(* Logix 5000 project; controller NSH_PLC1 vendor 1 type 14 code 167 rev 32.11; software revision 32.02 *)
// North State Hulling, PLC #1. Performes all System Logic and communicates with MCC#1, All Flex IO & PLC#2 (MCC#2 & #3)

TASK MainTask (continuous, watchdog 500 ms) : MainProgram, BagHouses, PreClean, HullerSheller

MODULES
   Local : vendor 1 type 14 code 167 (ICP 0, Ethernet 192.168.1.250, rev 32.11)
      AOP_BH1A : PowerFlex 755-EENET (Ethernet 192.168.0.41, rev 14.4, Output RPI 250 ms)   // Baghouse #1 Fan
          : vendor 1 type 143 code 32928 (RhinoBP 13, rev 1.1)
          : vendor 1 type 143 code 33184 (RhinoBP 14, rev 2.5)
      AOP_H28_D : PowerFlex 525-EENET (Ethernet 192.168.1.56, rev 6.1, Output RPI 250 ms)   // Nolan Shear Roll
      AOP_Local_Flex_IO : 1794-AENTR (Ethernet 192.168.0.32, rev 1.1, Output RPI 250 ms)   // PLC Panel Flex IO
         Input_L1 : 1794-IA16 (Flex 0, rev 1.1)
         Output_L6 : vendor 1 type 7 code 48 (Flex 5, rev 1.1)
         Input_L4 : 1794-IA16 (Flex 3, rev 1.1)
         Input_L5 : 1794-IA16 (Flex 4, rev 1.1)
         Input_L2 : 1794-IA16 (Flex 1, rev 1.1)
         Input_L3 : 1794-IA16 (Flex 2, rev 1.1)
         Output_L7 : vendor 1 type 7 code 48 (Flex 6, rev 1.1)
         Output_L8 : vendor 1 type 7 code 48 (Flex 7, rev 1.1)
      AOP_Remote_Flex_IO : 1794-AENTR (Ethernet 192.168.0.51, rev 1.1, Output RPI 250 ms)   // Remote Flex IO
         Input_R1 : 1794-IA16 (Flex 0, rev 1.1)
         Input_R2 : 1794-IA16 (Flex 1, rev 1.1)
         Input_R3 : 1794-IA16 (Flex 2, rev 1.1)
         Input_R4 : 1794-IA16 (Flex 3, rev 1.1)
         Input_R5 : 1794-IA16 (Flex 4, rev 1.1)
         Output_R6 : vendor 1 type 7 code 48 (Flex 5, rev 1.1)
         Output_R7 : vendor 1 type 7 code 48 (Flex 6, rev 1.1)
         Output_R8 : vendor 1 type 7 code 48 (Flex 7, rev 1.1)
      AOP_P_9A : 193-ECM-ETR (Ethernet 192.168.1.45, rev 7.1, StandardDataDriven RPI 250 ms)
END_MODULES

TYPE MainBins :   // Main Bins, Gates, Switches and Bindicators
STRUCT
   SW_A_Opened : BOOL;   // Line 1, Bin Gate Opened Switch
   SW_A_Closed : BOOL;   // Line 1, Bin Gate Closed Switch
   SV_Open_A : BOOL;   // Line 1, Open Bin Gate Soleniod
   SW_B_Opened : BOOL;   // Line 2, Bin Gate Opened Switch
   SW_B_Closed : BOOL;   // Line 2, Bin Gate Closed Switch
   SV_Open_B : BOOL;   // Line 2, Open Bin Gate Soleniod
   BN_Full : BOOL;   // Bin Full Bindicator
   TMR_BinFull : TIMER;   // Bin is Full TON Timer
   TMR_BinNotFull : TIMER;   // Bin is Not Full TON Timer
   LT_FullVisible : BOOL;   // HMI Bin Full Light, Visible
   LT_FullFlash : BOOL;   // HMI Bin Full Light, Flash
   MSG_Status_A : DINT;   // 0=Closed (Red) 1=Opened (Green) 2=Inbetween (Flash Yellow)
   MSG_Status_B : DINT;   // 0=Closed (Red) 1=Opened (Green) 2=Inbetween (Flash Yellow)
END_STRUCT
END_TYPE

TYPE Motor :
STRUCT
   StatusBits : DINT;   // Status Bits
   Run : BOOL;   // Run Motor
   Running : BOOL;   // Motor is Running
   NextMotorOK : BOOL;   // Ok, Run Next Motor
   Run_TON : TIMER;   // Running + Time, Run Next Motor
   Amps : REAL;   // Amps
   MSG_GraphicsState : DINT;   // 0=Red 1=Grn 2=FlashYel 3=FlashBlue 4=FlashRed
   HandAuto : BOOL;   // Radio Buttons, On=Hand, Off=Auto
   RunStop : BOOL;   // Pushbuttons, On=Run, Off=Stop
   Fault : BOOL;   // On=Fault
   Fault_TON : TIMER;   // Delay Before Fault
   Warning : BOOL;   // On=Warning
   Warning_TON : TIMER;   // Delay Before Warning
   MSG_FaultWarning : DINT;   // Display of Fault or Warning Number
   Reset_TOF : TIMER;   // Fault Reset Duration to Drive
   HandAuto_OSB : BOOL;   // Radio Buttons HandAuto Transition Relay
   DD_OverloadPercent : DINT;   // Overload 0.0-100.0%, Data Display
   StopTimer : TIMER;   // Shutdown Stop Timer
END_STRUCT
END_TYPE

TYPE VFD_Extra :
STRUCT
   DE_Speed : DINT;   // Speed, 1-100%, Data Entry
   DD_SpeedFactored : DINT;   // Speed, (1-100%, X Factor) Data Display
   DE_OverloadPercent : DINT;   // Overload Warning 1-100%, Data Entry
END_STRUCT
END_TYPE

VAR_GLOBAL   (* controller tags *)
   AFI : BOOL;   // Always False
   BH1 : Motor := (Run_TON.PRE := 1500, StopTimer.PRE := 1500);   // Auger
   BH1A : Motor := (Run_TON.PRE := 1500, StopTimer.PRE := 1500);   // Fan
   BH1A_VFD : VFD_Extra;   // Fan
   BH1B : Motor := (Run_TON.PRE := 1500, StopTimer.PRE := 1500);   // Rev.Fan
   BH1C : Motor := (Run_TON.PRE := 1500, StopTimer.PRE := 1500);   // Rev. Arm
   BH1D : Motor := (Run_TON.PRE := 1500, StopTimer.PRE := 1500);   // Airlock
   BH2 : Motor := (Run_TON.PRE := 1500, StopTimer.PRE := 1500);   // S. Ele
   BH2A : Motor := (Run_TON.PRE := 1500, StopTimer.PRE := 1500);   // Fan
   BH2A_VFD : VFD_Extra;   // Fan
   BH2B : Motor := (Run_TON.PRE := 1500, StopTimer.PRE := 1500);   // Rev.Fan
   BH2C : Motor := (Run_TON.PRE := 1500, StopTimer.PRE := 1500);   // Rev. Arm
   BH2D : Motor := (Run_TON.PRE := 1500);   // Airlock
   BH3 : Motor := (Run_TON.PRE := 1500, StopTimer.PRE := 1500);   // BH Rock
   BH3A : Motor := (Run_TON.PRE := 1500, StopTimer.PRE := 1500);   // Fan
   BH3A_VFD : VFD_Extra;   // Fan
   BH3B : Motor := (Run_TON.PRE := 1500, StopTimer.PRE := 1500);   // Rev.Fan
   BH3C : Motor := (Run_TON.PRE := 1500, StopTimer.PRE := 1500);   // Rev. Arm
   BH3D : Motor := (Run_TON.PRE := 1500, StopTimer.PRE := 1500);   // Airlock
   BH_FansStarting : BOOL;   // Baghouse 1, 2 or 3 Fans Starting
   C10 : Motor := (Run_TON.PRE := 1500, StopTimer.PRE := 1500);   // Auger
   C1A : Motor := (Run_TON.PRE := 1500, StopTimer.PRE := 1500);   // Auger
   C1B : Motor := (Run_TON.PRE := 1500, StopTimer.PRE := 1500);   // Auger
   C2 : Motor := (Run_TON.PRE := 1500, StopTimer.PRE := 1500);   // Auger
   C3A : Motor := (Run_TON.PRE := 1500, StopTimer.PRE := 1500);   // Auger
   C3B : Motor := (Run_TON.PRE := 1500, StopTimer.PRE := 1500);   // Auger
   C4 : Motor := (Run_TON.PRE := 1500, StopTimer.PRE := 1500);   // Ele.
   C5 : Motor := (Run_TON.PRE := 1500);   // Aspirator
   C7 : Motor := (Run_TON.PRE := 1500, StopTimer.PRE := 1500);   // Ele
   C8 : Motor := (Run_TON.PRE := 1500, StopTimer.PRE := 1500);   // Auger
   C9 : Motor := (Run_TON.PRE := 1500, StopTimer.PRE := 1500);   // Auger
   CL1 : Motor := (Run_TON.PRE := 1500, StopTimer.PRE := 1500);   // Auger
   CL2 : Motor := (Run_TON.PRE := 1500, StopTimer.PRE := 1500);   // Auger
   CL3 : Motor := (Run_TON.PRE := 1500, StopTimer.PRE := 1500);   // Auger
   CL4 : Motor := (Run_TON.PRE := 1500, StopTimer.PRE := 1500);   // Auger
   CL5 : Motor := (Run_TON.PRE := 1500, StopTimer.PRE := 1500);   // Auger
   CL6 : Motor := (Run_TON.PRE := 1500, StopTimer.PRE := 1500);   // Auger
   CR_LastBH1Fan : BOOL;   // Last Motor in Baghouse 1 Fans Running
   CR_LastBH2Fan : BOOL;   // Last Motor in Baghouse 2 Fans Running
   CR_LastBH3Fan : BOOL;   // Last Motor in Baghouse 3 Fans Running
   CR_LastLine1 : BOOL;   // Last Motor in line 1 Running
   CR_LastLine2 : BOOL;   // Last Motor in line 2 Running
   CR_LastPC1Fan : BOOL;   // Last Motor in Line 1 Fans Running
   CR_LastPC2Fan : BOOL;   // Last Motor in Line 2 Fans Running
   CR_RunBH2_Fans : BOOL;   // Run Baghouse 2 Fans Relay
   CR_RunBH2_FansCO : BOOL;   // Run Baghouse 2 Fans Cleanout Relay
   CR_RunBH3_Fans : BOOL;   // Run Baghouse 3 Fans Relay
   CR_RunBH3_FansCO : BOOL;   // Run Baghouse 3 Fans Cleanout Relay
   CR_RunBH_Fans : BOOL;   // Run Baghouse's Fans Relay
   CR_RunBH_FansCO : BOOL;   // Run Baghouse's Cleanout Relay
   CR_RunCommon : BOOL;   // PreClean, Run Common Units
   CR_RunHS : BOOL;   // Run Hullers & Shellers Relay
   CR_RunHullerShellers : BOOL;   // Run Hullers & Shellers
   CR_RunLine1 : BOOL;   // Pre Clean Run Line 1 Relay
   CR_RunLine2 : BOOL;   // Pre Clean Run Line 2 Relay
   CR_RunPC1_Fans : BOOL;   // Pre Clean Run Line 1 Fans Relay
   CR_RunPC1_FansCO : BOOL;   // Pre Clean Run Line 1 Fans Cleanout Relay
   CR_RunPC2_Fans : BOOL;   // Pre Clean Run Line 2 Fans Relay
   CR_RunPC2_FansCO : BOOL;   // Pre Clean Run Line 2 Fans Cleanout Relay
   CR_StopBH_Fans : BOOL;   // Stop Baghouse's Fans Relay
   CR_StopBH_FansCO : BOOL;   // Stop Baghouse's Fans Cleanout Relay
   CR_StopCommon : BOOL;   // PreClean, Stop Common Units
   CR_StopHS : BOOL;   // Stop Hullers & Shellers Relay
   CR_StopLine1 : BOOL;   // Pre Clean Stop Line 1 Relay
   CR_StopLine2 : BOOL;   // Pre Clean Stop Line 2 Relay
   CR_StopPC1_Fans : BOOL;   // Pre Clean Stop Line 1 Fans Relay
   CR_StopPC1_FansCO : BOOL;   // Pre Clean Stop Line 1 Fans Cleanout Relay
   CR_StopPC2_Fans : BOOL;   // Pre Clean Stop Line 2 Fans Relay
   CR_StopPC2_FansCO : BOOL;   // Pre Clean Stop Line 2 Fans Cleanout Relay
   D10 : Motor := (Run_TON.PRE := 1500, StopTimer.PRE := 1500);   // Ele
   D11 : Motor := (Run_TON.PRE := 1500, StopTimer.PRE := 1500);   // Auger
   D12 : Motor := (Run_TON.PRE := 1500, StopTimer.PRE := 1500);   // Auger
   D13 : Motor := (Run_TON.PRE := 1500, StopTimer.PRE := 1500);   // Auger
   D14 : Motor := (Run_TON.PRE := 1500, StopTimer.PRE := 1500);   // Auger
   D1A : Motor := (Run_TON.PRE := 1500, StopTimer.PRE := 1500);   // Auger
   D1B : Motor := (Run_TON.PRE := 1500, StopTimer.PRE := 1500);   // Auger
   D2 : Motor := (Run_TON.PRE := 1500, StopTimer.PRE := 1500);   // Auger
   D3 : Motor := (Run_TON.PRE := 1500);   // Aspirator
   D4 : Motor := (Run_TON.PRE := 1500, StopTimer.PRE := 1500);   // Auger
   D5 : Motor := (Run_TON.PRE := 1500, StopTimer.PRE := 1500);   // Auger
   D6 : Motor := (Run_TON.PRE := 1500, StopTimer.PRE := 1500);   // Auger
   D7 : Motor := (Run_TON.PRE := 1500);   // Aspirator
   DE_PC_MasterSpeedFactor : DINT;   // PreClean Master Speed Factor 75%->125%
   DL1 : Motor := (Run_TON.PRE := 1500, StopTimer.PRE := 1500);   // Auger
   DummyLastMotor : BOOL;   // Last Motor in Start Sequence
   DummyOutput : BOOL;
   DummyVFD : VFD_Extra;   // Dummy
   H1 : Motor := (Run_TON.PRE := 1500, StopTimer.PRE := 1500);   // Conv.
   H10 : Motor := (Run_TON.PRE := 1500, StopTimer.PRE := 1500);   // Auger
   H11 : Motor := (Run_TON.PRE := 1500, StopTimer.PRE := 1500);   // Ele.
   H12 : Motor := (Run_TON.PRE := 1500, StopTimer.PRE := 1500);   // Auger
   H13 : Motor := (Run_TON.PRE := 1500, StopTimer.PRE := 1500);   // Auger
   H14A : Motor := (Run_TON.PRE := 1500, StopTimer.PRE := 1500);   // Shr. Roll
   H14B : Motor := (Run_TON.PRE := 1500, StopTimer.PRE := 1500);   // Shr. Roll
   H14C : Motor := (Run_TON.PRE := 1500, StopTimer.PRE := 1500);   // Vib.
   H15A : Motor := (Run_TON.PRE := 1500, StopTimer.PRE := 1500);   // Aspirator
   H15B : Motor := (Run_TON.PRE := 1500, StopTimer.PRE := 1500);   // Aspirator
   H16 : Motor := (Run_TON.PRE := 1500, StopTimer.PRE := 1500);   // Auger
   H17 : Motor := (Run_TON.PRE := 1500, StopTimer.PRE := 1500);   // Roll Fd.
   H18A : Motor := (Run_TON.PRE := 1500, StopTimer.PRE := 1500);   // Shr. Roll
   H18B : Motor := (Run_TON.PRE := 1500, StopTimer.PRE := 1500);   // Shr. Roll
   H18C : Motor := (Run_TON.PRE := 1500, StopTimer.PRE := 1500);   // Vib.
   H19A : Motor := (Run_TON.PRE := 1500, StopTimer.PRE := 1500);   // Aspirator
   H19B : Motor := (Run_TON.PRE := 1500, StopTimer.PRE := 1500);   // Aspirator
   H20A : Motor := (Run_TON.PRE := 1500, StopTimer.PRE := 1500);   // Shr. Roll
   H20B : Motor := (Run_TON.PRE := 1500, StopTimer.PRE := 1500);   // Shr. Roll
   H20C : Motor := (Run_TON.PRE := 1500, StopTimer.PRE := 1500);   // Vib.
   H21A : Motor := (Run_TON.PRE := 1500, StopTimer.PRE := 1500);   // Aspirator
   H21B : Motor := (Run_TON.PRE := 1500, StopTimer.PRE := 1500);   // Aspirator
   H22 : Motor := (Run_TON.PRE := 1500, StopTimer.PRE := 1500);   // BMM
   H22B : Motor := (Run_TON.PRE := 1500);   // Hard Crkr.
   H23A : Motor := (Run_TON.PRE := 1500, StopTimer.PRE := 1500);   // Aspirator
   H23B : Motor := (Run_TON.PRE := 1500, StopTimer.PRE := 1500);   // Aspirator
   H24A : Motor := (Run_TON.PRE := 1500, StopTimer.PRE := 1500);   // Aspirator
   H24B : Motor := (Run_TON.PRE := 1500, StopTimer.PRE := 1500);   // Aspirator
   H25 : Motor := (Run_TON.PRE := 1500, StopTimer.PRE := 1500);   // Ele.
   H26 : Motor := (Run_TON.PRE := 1500, StopTimer.PRE := 1500);   // Auger
   H27 : Motor := (Run_TON.PRE := 1500, StopTimer.PRE := 1500);   // Auger
   H28A : Motor := (Run_TON.PRE := 1500, StopTimer.PRE := 1500);   // HC Vib.
   H28B : Motor := (Run_TON.PRE := 1500, StopTimer.PRE := 1500);   // Hard Crkr.
   H28C : Motor := (Run_TON.PRE := 1500, StopTimer.PRE := 1500);   // S.Roll
   H28D : Motor := (Run_TON.PRE := 1500, StopTimer.PRE := 1500);   // Shr.Roll.
   H29A : Motor := (Run_TON.PRE := 1500, StopTimer.PRE := 1500);   // Aspirator
   H29B : Motor := (Run_TON.PRE := 1500, StopTimer.PRE := 1500);   // Aspirator
   H30 : Motor := (Run_TON.PRE := 1500, StopTimer.PRE := 1500);   // Auger
   H31 : Motor := (Run_TON.PRE := 1500, StopTimer.PRE := 1500);   // Roll Fdr.
   H32A : Motor := (Run_TON.PRE := 1500, StopTimer.PRE := 1500);   // HS Cracker
   H32B : Motor := (Run_TON.PRE := 1500, StopTimer.PRE := 1500);   // Hard Crkr.
   H32C : Motor := (Run_TON.PRE := 1500, StopTimer.PRE := 1500);   // Shr.Roll.
   H32D : Motor := (Run_TON.PRE := 1500, StopTimer.PRE := 1500);   // Shr.Roll.
   H33A : Motor := (Run_TON.PRE := 1500, StopTimer.PRE := 1500);   // Aspirator
   H33B : Motor := (Run_TON.PRE := 1500, StopTimer.PRE := 1500);   // Aspirator
   H34A : Motor := (Run_TON.PRE := 1500, StopTimer.PRE := 1500);   // HC Vib.
   H34B : Motor := (Run_TON.PRE := 1500, StopTimer.PRE := 1500);   // Hard Crkr.
   H34C : Motor := (Run_TON.PRE := 1500, StopTimer.PRE := 1500);   // S.Roll
   H34D : Motor := (Run_TON.PRE := 1500, StopTimer.PRE := 1500);   // Shr.Roll.
   H35A : Motor := (Run_TON.PRE := 1500, StopTimer.PRE := 1500);   // Aspirator
   H35B : Motor := (Run_TON.PRE := 1500, StopTimer.PRE := 1500);   // Aspirator
   H36 : Motor := (Run_TON.PRE := 1500, StopTimer.PRE := 1500);   // BMM
   H37A : Motor := (Run_TON.PRE := 1500, StopTimer.PRE := 1500);   // Aspirator
   H37B : Motor := (Run_TON.PRE := 1500, StopTimer.PRE := 1500);   // Aspirator
   H38A : Motor := (Run_TON.PRE := 1500, StopTimer.PRE := 1500);   // Aspirator
   H38B : Motor := (Run_TON.PRE := 1500, StopTimer.PRE := 1500);   // Aspirator
   H39 : Motor := (Run_TON.PRE := 1500, StopTimer.PRE := 1500);   // Ele.
   H3A : Motor := (Run_TON.PRE := 1500, StopTimer.PRE := 1500);   // Incline
   H3B : Motor := (Run_TON.PRE := 1500, StopTimer.PRE := 1500);   // Ele.
   H4 : Motor := (Run_TON.PRE := 1500, StopTimer.PRE := 1500);   // Auger
   H40 : Motor := (Run_TON.PRE := 1500, StopTimer.PRE := 1500);   // Auger
   H41 : Motor := (Run_TON.PRE := 1500, StopTimer.PRE := 1500);   // Auger
   H42A : Motor := (Run_TON.PRE := 1500, StopTimer.PRE := 1500);   // HC Vib.
   H42B : Motor := (Run_TON.PRE := 1500, StopTimer.PRE := 1500);   // Hard Crkr.
   H42C : Motor := (Run_TON.PRE := 1500, StopTimer.PRE := 1500);   // S.Roll
   H42D : Motor := (Run_TON.PRE := 1500, StopTimer.PRE := 1500);   // Shr.Roll.
   H42H : Motor := (Run_TON.PRE := 1500);   // Auger
   H43A : Motor := (Run_TON.PRE := 1500, StopTimer.PRE := 1500);   // Aspirator
   H43B : Motor := (Run_TON.PRE := 1500, StopTimer.PRE := 1500);   // Aspirator
   H44A : Motor := (Run_TON.PRE := 1500, StopTimer.PRE := 1500);   // HC Vib.
   H44B : Motor := (Run_TON.PRE := 1500, StopTimer.PRE := 1500);   // Hard Crkr.
   H44C : Motor := (Run_TON.PRE := 1500, StopTimer.PRE := 1500);   // S.Roll
   H44D : Motor := (Run_TON.PRE := 1500, StopTimer.PRE := 1500);   // Shr.Roll.
   H45A : Motor := (Run_TON.PRE := 1500, StopTimer.PRE := 1500);   // Aspirator
   H45B : Motor := (Run_TON.PRE := 1500, StopTimer.PRE := 1500);   // Aspirator
   H46 : Motor := (Run_TON.PRE := 1500, StopTimer.PRE := 1500);   // BMM
   H47A : Motor := (Run_TON.PRE := 1500, StopTimer.PRE := 1500);   // Aspirator
   H47B : Motor := (Run_TON.PRE := 1500, StopTimer.PRE := 1500);   // Aspirator
   H48A : Motor := (Run_TON.PRE := 1500, StopTimer.PRE := 1500);   // Aspirator
   H48B : Motor := (Run_TON.PRE := 1500, StopTimer.PRE := 1500);   // Aspirator
   H49 : Motor := (Run_TON.PRE := 1500, StopTimer.PRE := 1500);   // Ele.
   H5 : Motor := (Run_TON.PRE := 1500, StopTimer.PRE := 1500);   // Auger
   H50A : Motor := (Run_TON.PRE := 1500, StopTimer.PRE := 1500);   // Auger
   H50B : Motor := (Run_TON.PRE := 1500, StopTimer.PRE := 1500);   // Auger
   H6 : Motor := (Run_TON.PRE := 1500, StopTimer.PRE := 1500);   // Roll Fd.
   H7 : Motor := (Run_TON.PRE := 1500, StopTimer.PRE := 1500);   // BMM
   H8A : Motor := (Run_TON.PRE := 1500, StopTimer.PRE := 1500);   // Aspirator
   H8B : Motor := (Run_TON.PRE := 1500, StopTimer.PRE := 1500);   // Aspirator
   H9A : Motor := (Run_TON.PRE := 1500, StopTimer.PRE := 1500);   // Aspirator
   H9B : Motor := (Run_TON.PRE := 1500, StopTimer.PRE := 1500);   // Aspirator
   HS_Horn : BOOL;   // Huller Sheller, Horn Output
   HS_LastMotor : BOOL;   // Last Motor in Huller Sheller Sequence is Running
   HS_NoEstops : BOOL;   // Huller Sheller, No Estops
   HS_Starting : BOOL;   // Sheller Sequence is Starting, Prevent Preclean from Starting
   LS101 : BOOL;   // Dummy Limit Switch
   M10 : Motor := (Run_TON.PRE := 1500, StopTimer.PRE := 1500);   // Vib.
   M10A : Motor := (Run_TON.PRE := 1500, StopTimer.PRE := 1500);   // Asp.
   M10B : Motor := (Run_TON.PRE := 1500, StopTimer.PRE := 1500);   // Asp.
   M11 : Motor := (Run_TON.PRE := 1500, StopTimer.PRE := 1500);   // Ele.
   M12aA : Motor := (Run_TON.PRE := 1500, StopTimer.PRE := 1500);   // Grav.Sep
   M12aB : Motor := (Run_TON.PRE := 1500, StopTimer.PRE := 1500);   // Syntron
   M13aA : Motor := (Run_TON.PRE := 1500, StopTimer.PRE := 1500);   // Grav.Sep
   M13aB : Motor := (Run_TON.PRE := 1500, StopTimer.PRE := 1500);   // Syntron
   M14 : Motor := (Run_TON.PRE := 1500, StopTimer.PRE := 1500);   // Vib.
   M15 : Motor := (Run_TON.PRE := 1500, StopTimer.PRE := 1500);   // Ele.
   M16 : Motor := (Run_TON.PRE := 1500, StopTimer.PRE := 1500);   // Evo.
   M16R : Motor;   // Conveyor
   M17 : Motor := (Run_TON.PRE := 1500, StopTimer.PRE := 1500);   // Evo.
   M18 : Motor := (Run_TON.PRE := 1500, StopTimer.PRE := 1500);   // Vib.
   M19 : Motor := (Run_TON.PRE := 1500, StopTimer.PRE := 1500);   // Ele.
   M1A : Motor := (Run_TON.PRE := 1500, StopTimer.PRE := 1500);   // Vib.
   M2 : Motor := (Run_TON.PRE := 1500, StopTimer.PRE := 1500);   // Vib.
   M20 : Motor := (Run_TON.PRE := 1500, StopTimer.PRE := 1500);   // Ele.
   M21 : Motor := (Run_TON.PRE := 1500, StopTimer.PRE := 1500);   // Nolin
   M25 : Motor := (Run_TON.PRE := 1500, StopTimer.PRE := 1500);   // Accept Vib.
   M27 : Motor := (Run_TON.PRE := 1500, StopTimer.PRE := 1500);   // Belt
   M28 : Motor := (Run_TON.PRE := 1500, StopTimer.PRE := 1500);   // Belt
   M29 : Motor := (Run_TON.PRE := 1500, StopTimer.PRE := 1500);   // Ele.
   M3 : Motor := (Run_TON.PRE := 1500, StopTimer.PRE := 1500);   // Belt
   M30A : Motor := (Run_TON.PRE := 1500, StopTimer.PRE := 1500);   // HC Vib.
   M30B : Motor := (Run_TON.PRE := 1500, StopTimer.PRE := 1500);   // Hard Crkr.
   M30C : Motor := (Run_TON.PRE := 1500, StopTimer.PRE := 1500);   // Shr.Roll.
   M30D : Motor := (Run_TON.PRE := 1500, StopTimer.PRE := 1500);   // Shr.Roll.
   M31A : Motor := (Run_TON.PRE := 1500, StopTimer.PRE := 1500);   // Asp.
   M31B : Motor := (Run_TON.PRE := 1500, StopTimer.PRE := 1500);   // Asp.
   M32A : Motor := (Run_TON.PRE := 1500, StopTimer.PRE := 1500);   // Vib.Scrn.
   M32B : Motor := (Run_TON.PRE := 1500, StopTimer.PRE := 1500);   // Ele.
   M33 : Motor := (Run_TON.PRE := 1500, StopTimer.PRE := 1500);   // Belt
   M34 : Motor := (Run_TON.PRE := 1500, StopTimer.PRE := 1500);   // Destoner
   M35 : Motor := (Run_TON.PRE := 1500, StopTimer.PRE := 1500);   // Ele.
   M36A : Motor := (Run_TON.PRE := 1500, StopTimer.PRE := 1500);   // G. Sep.
   M36B : Motor := (Run_TON.PRE := 1500, StopTimer.PRE := 1500);   // R. Feeder.
   M37 : Motor := (Run_TON.PRE := 1500, StopTimer.PRE := 1500);   // 5x12
   M38A : Motor := (Run_TON.PRE := 1500, StopTimer.PRE := 1500);   // Asp.
   M38B : Motor := (Run_TON.PRE := 1500, StopTimer.PRE := 1500);   // Asp.
   M39 : Motor := (Run_TON.PRE := 1500, StopTimer.PRE := 1500);   // Ele.
   M391 : Motor := (Run_TON.PRE := 1500);   // Ele.
   M4 : Motor := (Run_TON.PRE := 1500, StopTimer.PRE := 1500);   // Vib.
   M40A : Motor := (Run_TON.PRE := 1500, StopTimer.PRE := 1500);   // Sep.
   M40B : Motor := (Run_TON.PRE := 1500, StopTimer.PRE := 1500);   // Syn.Fer.
   M41 : Motor := (Run_TON.PRE := 1500, StopTimer.PRE := 1500);   // Ele.
   M42C : Motor := (Run_TON.PRE := 1500, StopTimer.PRE := 1500);   // 3C Deck
   M42D : Motor := (Run_TON.PRE := 1500, StopTimer.PRE := 1500);   // 3C Deck
   M43CA : Motor := (Run_TON.PRE := 1500, StopTimer.PRE := 1500);   // Asp.
   M43CB : Motor := (Run_TON.PRE := 1500, StopTimer.PRE := 1500);   // Asp.
   M43DA : Motor := (Run_TON.PRE := 1500, StopTimer.PRE := 1500);   // Asp.
   M43DB : Motor := (Run_TON.PRE := 1500, StopTimer.PRE := 1500);   // Asp.
   M44A : Motor := (Run_TON.PRE := 1500, StopTimer.PRE := 1500);   // Belt
   M44B : Motor := (Run_TON.PRE := 1500, StopTimer.PRE := 1500);   // Belt
   M5 : Motor := (Run_TON.PRE := 1500, StopTimer.PRE := 1500);   // Vib.
   M6 : Motor := (Run_TON.PRE := 1500, StopTimer.PRE := 1500);   // Belt
   M7 : Motor := (Run_TON.PRE := 1500, StopTimer.PRE := 1500);   // Ele.
   M8 : Motor := (Run_TON.PRE := 1500, StopTimer.PRE := 1500);   // Shkr.
   M9A : Motor := (Run_TON.PRE := 1500, StopTimer.PRE := 1500);   // Asp.
   M9B : Motor := (Run_TON.PRE := 1500, StopTimer.PRE := 1500);   // Asp.
   MainBin1 : MainBins;   // PreClean to Huller, Main Bin #1
   MainBin2 : MainBins;   // PreClean to Huller, Main Bin #1
   MainBin3 : MainBins;   // PreClean to Huller, Main Bin #1
   MainBin4 : MainBins;   // PreClean to Huller, Main Bin #1
   MainBin5 : MainBins;   // PreClean to Huller, Main Bin #1
   MainBin6 : MainBins;   // PreClean to Huller, Main Bin #1
   MainBin7 : MainBins;   // PreClean to Huller, Main Bin #1
   MainBin8 : MainBins;   // PreClean to Huller, Main Bin #1
   NewWarning : BOOL;   // New Huller-Sheller Warning has just occured
   Num_Warning_LS : DINT;   // Number of Warnings Last Scan, Detect New
   P10_5A : Motor := (Run_TON.PRE := 1500, StopTimer.PRE := 1500);   // Cross Auger
   P10_5B : Motor := (Run_TON.PRE := 1500, StopTimer.PRE := 1500);   // Cross Auger
   P10A : Motor := (Run_TON.PRE := 1500, StopTimer.PRE := 1500);   // Elev to Bins
   P10B : Motor := (Run_TON.PRE := 1500, StopTimer.PRE := 1500);   // Elev to Bins
   P11A : Motor := (Run_TON.PRE := 1500, StopTimer.PRE := 1500);   // Line1 Auger
   P11B : Motor := (Run_TON.PRE := 1500, StopTimer.PRE := 1500);   // Line2 Auger
   P1A : Motor := (Run_TON.PRE := 1500, StopTimer.PRE := 1500);   // DO Conv.
   P1B : Motor := (Run_TON.PRE := 1500, StopTimer.PRE := 1500);   // Auger
   P2A : Motor := (Run_TON.PRE := 1500, StopTimer.PRE := 1500);   // Cross Conv.
   P2B : Motor := (Run_TON.PRE := 1500, StopTimer.PRE := 1500);   // Stick Reel
   P3A : Motor := (Run_TON.PRE := 1500, StopTimer.PRE := 1500);   // Stick Reel
   P3B : Motor := (Run_TON.PRE := 1500, StopTimer.PRE := 1500);   // Stick Reel
   P4A : Motor := (Run_TON.PRE := 1500, StopTimer.PRE := 1500);   // C. Belt
   P4B : Motor := (Run_TON.PRE := 1500, StopTimer.PRE := 1500);   // C. Belt
   P5A : Motor := (Run_TON.PRE := 1500, StopTimer.PRE := 1500);   // Ele. to Vib
   P5B : Motor := (Run_TON.PRE := 1500, StopTimer.PRE := 1500);   // Ele. to Vib
   P6A : Motor := (Run_TON.PRE := 1500, StopTimer.PRE := 1500);   // Vib Splitter
   P6B : Motor := (Run_TON.PRE := 1500, StopTimer.PRE := 1500);   // Vib.Spltr.
   P7A : Motor := (Run_TON.PRE := 1500, StopTimer.PRE := 1500);   // Screener
   P7A1 : Motor := (Run_TON.PRE := 1500);   // Screener
   P7A2 : Motor := (Run_TON.PRE := 1500, StopTimer.PRE := 1500);   // Screener
   P7B : Motor := (Run_TON.PRE := 1500, StopTimer.PRE := 1500);   // Screener
   P7B2_A : Motor := (Run_TON.PRE := 1500, StopTimer.PRE := 1500);   // Screener
   P7B2_B : Motor := (Run_TON.PRE := 1500, StopTimer.PRE := 1500);   // Rot.Fdr.
   P8A2_A : Motor := (Run_TON.PRE := 1500, StopTimer.PRE := 1500);   // Destoner
   P8A2_B : Motor := (Run_TON.PRE := 1500, StopTimer.PRE := 1500);   // AirLock
   P8A_A : Motor := (Run_TON.PRE := 1500, StopTimer.PRE := 1500);   // Destoner
   P8A_B : Motor := (Run_TON.PRE := 1500, StopTimer.PRE := 1500);   // Airlock
   P8B : Motor := (Run_TON.PRE := 1500, StopTimer.PRE := 1500);   // Destoner
   P8B2_A : Motor := (Run_TON.PRE := 1500, StopTimer.PRE := 1500);   // Destoner
   P8B2_B : Motor := (Run_TON.PRE := 1500, StopTimer.PRE := 1500);   // Rot.Fdr.
   P9A : Motor := (Run_TON.PRE := 1500, StopTimer.PRE := 1500);   // Auger
   P9B : Motor := (Run_TON.PRE := 1500, StopTimer.PRE := 1500);   // Auger
   PB_HS_Inshell : BOOL;   // Hullers & Shellers Run Inshell Button
   PB_HS_Meats : BOOL;   // Hullers & Shellers Run Meats Button
   PB_HSFaultReset : BOOL;   // Huller Sheller, Fault Reset Button
   PB_PCFaultReset : BOOL;   // PreClean Fault Reset Button
   PB_StartBH_Fans : BOOL;   // Start Baghouse's Fans Button
   PB_StartBH_FansCO : BOOL;   // Start Baghouse's Cleanout Button
   PB_StartHS : BOOL;   // Start Hullers & Shellers Button
   PB_StartLine1 : BOOL;   // Pre Clean Start Line 1 Button
   PB_StartLine2 : BOOL;   // Pre Clean Start Line 2 Button
   PB_StartPC1_Fans : BOOL;   // Pre Clean Start Line 1 Fans Button
   PB_StartPC1_FansCO : BOOL;   // Pre Clean Start Line 1 Fans Cleanout Button
   PB_StartPC2_Fans : BOOL;   // Pre Clean Start Line 2 Fans Button
   PB_StartPC2_FansCO : BOOL;   // Pre Clean Start Line 2 Fans Cleanout Button
   PB_StopBH_Fans : BOOL;   // Stop Baghouse's Fans Button
   PB_StopBH_FansCO : BOOL;   // Stop Baghouse's Fans Cleanout Button
   PB_StopHS : BOOL;   // Stop Hullers & Shellers Button
   PB_StopLine1 : BOOL;   // Pre Clean Stop Line 1 Button
   PB_StopLine2 : BOOL;   // Pre Clean Stop Line 2 Button
   PB_StopPC1_Fans : BOOL;   // Pre Clean Stop Line 1 Fans Button
   PB_StopPC1_FansCO : BOOL;   // Pre Clean Stop Line 1 Fans Cleanout Button
   PB_StopPC2_Fans : BOOL;   // Pre Clean Stop Line 2 Fans Button
   PB_StopPC2_FansCO : BOOL;   // Pre Clean Stop Line 2 Fans Cleanout Button
   PBB1A : Motor := (Run_TON.PRE := 1500, StopTimer.PRE := 1500);   // AirLock
   PBB1B : Motor := (Run_TON.PRE := 1500, StopTimer.PRE := 1500);   // Arm
   PBB1C : Motor := (Run_TON.PRE := 1500, StopTimer.PRE := 1500);   // Cleaning Fan,
   PBB1D : Motor := (Run_TON.PRE := 1500, StopTimer.PRE := 1500);   // Fan,
   PBB1D_VFD : VFD_Extra;   // Fan
   PBB2A : Motor := (Run_TON.PRE := 1500, StopTimer.PRE := 1500);   // AirLock
   PBB2B : Motor := (Run_TON.PRE := 1500, StopTimer.PRE := 1500);   // Arm
   PBB2C : Motor := (Run_TON.PRE := 1500, StopTimer.PRE := 1500);   // Cleaning Fan,
   PBB2D : Motor := (Run_TON.PRE := 1500, StopTimer.PRE := 1500);   // Fan,
   PBL_HS_Inshell : BOOL;   // Hullers & Shellers Run Inshell Button Light
   PBL_HS_Meats : BOOL;   // Hullers & Shellers Run Meats Button Light
   PBL_PCFaultReset : BOOL;   // PreClean Fault Reset Button Light
   PBL_StartBH_Fans : BOOL;   // Start Baghouse's Fans Button Light
   PBL_StartBH_FansCO : BOOL;   // Start Baghouse's Cleanout Button Light
   PBL_StartHS : BOOL;   // Start Hullers & Shellers Button Light
   PBL_StartLine1 : BOOL;   // Pre Clean Start Line 1 Button Light
   PBL_StartLine2 : BOOL;   // Pre Clean Start Line 2 Button Light
   PBL_StartPC1_Fans : BOOL;   // Pre Clean Start Line 1 Fans Button Light
   PBL_StartPC1_FansCO : BOOL;   // Pre Clean Start Line 1 Fans Cleanout Button Light
   PBL_StartPC2_Fans : BOOL;   // Pre Clean Start Line 2 Fans Button Light
   PBL_StartPC2_FansCO : BOOL;   // Pre Clean Start Line 2 Fans Cleanout Button Light
   PBL_StopBH_Fans : BOOL;   // Stop Baghouse's Fans Button Light
   PBL_StopBH_FansCO : BOOL;   // Stop Baghouse's Fans Cleanout Button Light
   PBL_StopHS : BOOL;   // Stop Hullers & Shellers Button Light
   PBL_StopLine1 : BOOL;   // Pre Clean Stop Line 1 Button Light
   PBL_StopLine2 : BOOL;   // Pre Clean Stop Line 2 Button Light
   PBL_StopPC1_Fans : BOOL;   // Pre Clean Stop Line 1 Fans Button Light
   PBL_StopPC1_FansCO : BOOL;   // Pre Clean Stop Line 1 Fans Cleanout Button Light
   PBL_StopPC2_Fans : BOOL;   // Pre Clean Stop Line 2 Fans Button Light
   PBL_StopPC2_FansCO : BOOL;   // Pre Clean Stop Line 2 Fans Cleanout Button Light
   PC_AlarmPulseHorn : BOOL;   // PreClean, New Alarm, Pulse Horn
   PC_FansStarting : BOOL;   // Pre Clean Fans Starting
   PC_FaultResetHorn : BOOL;   // PreClean, Fault Reset, sound Horn
   PC_Horn : BOOL;   // PreClean, Horn Output
   PC_LinesStarting : BOOL;   // Pre Clean Line 1 or 2 Starting
   PC_NoEstops : BOOL;   // PreClean, No Estops
   PD1 : Motor := (Run_TON.PRE := 1500, StopTimer.PRE := 1500);   // Dirt Conv.
   PD2 : Motor := (Run_TON.PRE := 1500, StopTimer.PRE := 1500);   // Incline
   PR1 : Motor := (Run_TON.PRE := 1500, StopTimer.PRE := 1500);   // Rock Conv.
   PR2 : Motor := (Run_TON.PRE := 1500, StopTimer.PRE := 1500);   // Inc. Rock
   PR3 : Motor := (Run_TON.PRE := 1500, StopTimer.PRE := 1500);   // Belt
   PS1 : Motor := (Run_TON.PRE := 1500, StopTimer.PRE := 1500);   // Stick Conv.
   PS2 : Motor := (Run_TON.PRE := 1500, StopTimer.PRE := 1500);   // Inc. Stick Conv.
   PS3 : Motor := (Run_TON.PRE := 1500, StopTimer.PRE := 1500);   // Twig Conv.
   PS4 : Motor := (Run_TON.PRE := 1500, StopTimer.PRE := 1500);   // Twig Conv.
   S1 : Motor := (Run_TON.PRE := 1500, StopTimer.PRE := 1500);   // Vib.
   S10 : Motor := (Run_TON.PRE := 1500, StopTimer.PRE := 1500);   // Auger
   S11 : Motor := (Run_TON.PRE := 1500, StopTimer.PRE := 1500);   // Ele.
   S12 : Motor := (Run_TON.PRE := 1500, StopTimer.PRE := 1500);   // Auger
   S13 : Motor := (Run_TON.PRE := 1500, StopTimer.PRE := 1500);   // Ele.
   S14 : Motor := (Run_TON.PRE := 1500, StopTimer.PRE := 1500);   // Auger
   S15 : Motor := (Run_TON.PRE := 1500, StopTimer.PRE := 1500);   // Auger
   S16A : Motor := (Run_TON.PRE := 1500, StopTimer.PRE := 1500);   // Auger
   S16B : Motor := (Run_TON.PRE := 1500, StopTimer.PRE := 1500);   // Auger
   S17A : Motor := (Run_TON.PRE := 1500, StopTimer.PRE := 1500);   // HS Cracker
   S17B : Motor := (Run_TON.PRE := 1500, StopTimer.PRE := 1500);   // Hard Crkr.
   S17C : Motor := (Run_TON.PRE := 1500, StopTimer.PRE := 1500);   // Shr.Roll.
   S17D : Motor := (Run_TON.PRE := 1500, StopTimer.PRE := 1500);   // S.Roll
   S18A : Motor := (Run_TON.PRE := 1500, StopTimer.PRE := 1500);   // HC Vib.
   S18B : Motor := (Run_TON.PRE := 1500, StopTimer.PRE := 1500);   // Hard Crkr.
   S18C : Motor := (Run_TON.PRE := 1500, StopTimer.PRE := 1500);   // Shr.Roll.
   S18D : Motor := (Run_TON.PRE := 1500, StopTimer.PRE := 1500);   // S.Roll
   S19 : Motor := (Run_TON.PRE := 1500, StopTimer.PRE := 1500);   // Gry.
   S2 : Motor := (Run_TON.PRE := 1500, StopTimer.PRE := 1500);   // Ele.
   S20 : Motor := (Run_TON.PRE := 1500, StopTimer.PRE := 1500);   // Ele.
   S21 : Motor := (Run_TON.PRE := 1500, StopTimer.PRE := 1500);   // Roll Fdr.
   S22A : Motor := (Run_TON.PRE := 1500, StopTimer.PRE := 1500);   // HC Vib.
   S22B : Motor := (Run_TON.PRE := 1500, StopTimer.PRE := 1500);   // Hard Crkr.
   S22C : Motor := (Run_TON.PRE := 1500, StopTimer.PRE := 1500);   // Shr.Roll.
   S22D : Motor := (Run_TON.PRE := 1500, StopTimer.PRE := 1500);   // S.Roll
   S23A : Motor := (Run_TON.PRE := 1500, StopTimer.PRE := 1500);   // HC Vib.
   S23B : Motor := (Run_TON.PRE := 1500, StopTimer.PRE := 1500);   // Hard Crkr.
   S23C : Motor := (Run_TON.PRE := 1500, StopTimer.PRE := 1500);   // Shr.Roll.
   S23D : Motor := (Run_TON.PRE := 1500, StopTimer.PRE := 1500);   // S.Roll
   S24 : Motor := (Run_TON.PRE := 1500, StopTimer.PRE := 1500);   // Deck
   S25 : Motor := (Run_TON.PRE := 1500, StopTimer.PRE := 1500);   // Ele.
   S26 : Motor := (Run_TON.PRE := 1500, StopTimer.PRE := 1500);   // Auger
   S27 : Motor := (Run_TON.PRE := 1500, StopTimer.PRE := 1500);   // Roll Fdr
   S28A : Motor := (Run_TON.PRE := 1500, StopTimer.PRE := 1500);   // HC Vib.
   S28B : Motor := (Run_TON.PRE := 1500, StopTimer.PRE := 1500);   // Hard Crkr.
   S28C : Motor := (Run_TON.PRE := 1500, StopTimer.PRE := 1500);   // Shr.Roll.
   S28D : Motor := (Run_TON.PRE := 1500, StopTimer.PRE := 1500);   // S.Roll
   S29A : Motor := (Run_TON.PRE := 1500, StopTimer.PRE := 1500);   // HC Vib.
   S29B : Motor := (Run_TON.PRE := 1500, StopTimer.PRE := 1500);   // Hard Crkr.
   S29C : Motor := (Run_TON.PRE := 1500, StopTimer.PRE := 1500);   // Shr.Roll.
   S29D : Motor := (Run_TON.PRE := 1500, StopTimer.PRE := 1500);   // S.Roll
   S3 : Motor := (Run_TON.PRE := 1500, StopTimer.PRE := 1500);   // Auger
   S30 : Motor := (Run_TON.PRE := 1500, StopTimer.PRE := 1500);   // Ele.
   S31 : Motor := (Run_TON.PRE := 1500, StopTimer.PRE := 1500);   // Auger
   S32A : Motor := (Run_TON.PRE := 1500, StopTimer.PRE := 1500);   // HC Vib.
   S32B : Motor := (Run_TON.PRE := 1500, StopTimer.PRE := 1500);   // Hard Crkr.
   S32C : Motor := (Run_TON.PRE := 1500, StopTimer.PRE := 1500);   // Shr.Roll.
   S32D : Motor := (Run_TON.PRE := 1500, StopTimer.PRE := 1500);   // S.Roll
   S33A : Motor := (Run_TON.PRE := 1500, StopTimer.PRE := 1500);   // HC Vib.
   S33B : Motor := (Run_TON.PRE := 1500, StopTimer.PRE := 1500);   // Hard Crkr.
   S33C : Motor := (Run_TON.PRE := 1500, StopTimer.PRE := 1500);   // Shr.Roll.
   S33D : Motor := (Run_TON.PRE := 1500, StopTimer.PRE := 1500);   // S.Roll
   S34 : Motor := (Run_TON.PRE := 1500, StopTimer.PRE := 1500);   // Deck
   S35 : Motor := (Run_TON.PRE := 1500, StopTimer.PRE := 1500);   // Ele.
   S36 : Motor := (Run_TON.PRE := 1500, StopTimer.PRE := 1500);   // Auger
   S37A : Motor := (Run_TON.PRE := 1500, StopTimer.PRE := 1500);   // HC Vib.
   S37B : Motor := (Run_TON.PRE := 1500, StopTimer.PRE := 1500);   // Hard Crkr.
   S37C : Motor := (Run_TON.PRE := 1500, StopTimer.PRE := 1500);   // Shr.Roll.
   S37D : Motor := (Run_TON.PRE := 1500, StopTimer.PRE := 1500);   // S.Roll
   S38 : Motor := (Run_TON.PRE := 1500, StopTimer.PRE := 1500);   // Shkr.
   S39 : Motor := (Run_TON.PRE := 1500, StopTimer.PRE := 1500);   // Ele.
   S40A : Motor := (Run_TON.PRE := 1500, StopTimer.PRE := 1500);   // HC Vib.
   S40B : Motor := (Run_TON.PRE := 1500, StopTimer.PRE := 1500);   // Hard Crkr.
   S40C : Motor := (Run_TON.PRE := 1500, StopTimer.PRE := 1500);   // Shr.Roll.
   S40D : Motor := (Run_TON.PRE := 1500, StopTimer.PRE := 1500);   // S.Roll
   S41 : Motor := (Run_TON.PRE := 1500, StopTimer.PRE := 1500);   // Ele.
   S42A : Motor := (Run_TON.PRE := 1500, StopTimer.PRE := 1500);   // HC Vib.
   S42B : Motor := (Run_TON.PRE := 1500, StopTimer.PRE := 1500);   // Hard Crkr.
   S42C : Motor := (Run_TON.PRE := 1500, StopTimer.PRE := 1500);   // S.Roll
   S42D : Motor := (Run_TON.PRE := 1500, StopTimer.PRE := 1500);   // Shr.Roll.
   S43 : Motor := (Run_TON.PRE := 1500, StopTimer.PRE := 1500);   // Shkr.
   S44 : Motor := (Run_TON.PRE := 1500, StopTimer.PRE := 1500);   // Ele.
   S45 : Motor := (Run_TON.PRE := 1500, StopTimer.PRE := 1500);   // Auger
   S46A : Motor := (Run_TON.PRE := 1500, StopTimer.PRE := 1500);   // HC Vib.
   S46B : Motor := (Run_TON.PRE := 1500, StopTimer.PRE := 1500);   // Hard Crkr.
   S46C : Motor := (Run_TON.PRE := 1500, StopTimer.PRE := 1500);   // S.Roll
   S46D : Motor := (Run_TON.PRE := 1500, StopTimer.PRE := 1500);   // Shr.Roll.
   S47 : Motor := (Run_TON.PRE := 1500, StopTimer.PRE := 1500);   // Auger
   S48 : Motor := (Run_TON.PRE := 1500, StopTimer.PRE := 1500);   // Auger
   S49 : Motor := (Run_TON.PRE := 1500, StopTimer.PRE := 1500);   // Auger
   S4A : Motor := (Run_TON.PRE := 1500, StopTimer.PRE := 1500);   // Aspirator
   S4B : Motor := (Run_TON.PRE := 1500, StopTimer.PRE := 1500);   // Aspirator
   S50 : Motor := (Run_TON.PRE := 1500, StopTimer.PRE := 1500);   // Auger
   S5A : Motor := (Run_TON.PRE := 1500, StopTimer.PRE := 1500);   // Aspirator
   S5B : Motor := (Run_TON.PRE := 1500, StopTimer.PRE := 1500);   // Aspirator
   S6 : Motor := (Run_TON.PRE := 1500, StopTimer.PRE := 1500);   // Belt
   S7 : Motor := (Run_TON.PRE := 1500, StopTimer.PRE := 1500);   // Ele.
   S8 : Motor := (Run_TON.PRE := 1500, StopTimer.PRE := 1500);   // Auger
   S9 : Motor := (Run_TON.PRE := 1500, StopTimer.PRE := 1500);   // Ele.
   SL1 : Motor := (Run_TON.PRE := 1500, StopTimer.PRE := 1500);   // Auger
   T1 : Motor := (Run_TON.PRE := 1500, StopTimer.PRE := 1500);   // Belt
   T2 : Motor := (Run_TON.PRE := 1500, StopTimer.PRE := 1500);   // Belt
   T3 : Motor := (Run_TON.PRE := 1500, StopTimer.PRE := 1500);   // Belt
   TMR_AutoStopBH_FansCO : TIMER := (PRE := 900000);   // Baghouse's Fans Auto Stop Clean Cleanout Timer
   TMR_AutoStopPC1_FansCO : TIMER := (PRE := 900000);   // Pre Clean Line 1 Fans Auto Stop Clean Cleanout Timer
   TMR_AutoStopPC2_FansCO : TIMER := (PRE := 900000);   // Pre Clean Line 2 Fans Auto Stop Clean Cleanout Timer
   TMR_FaultResetHorn : TIMER := (PRE := 3000);   // Fault Reset Sound Horn Duraton
   TMR_LineStart1 : TIMER := (PRE := 3000);   // Pre Clean Line 1 Start Warning Timer
   TMR_LineStart2 : TIMER := (PRE := 3000);   // Pre Clean Line 2 Start Warning Timer
   TMR_StartBH_Fans : TIMER := (PRE := 3000);   // Start Baghouse's Fans Timer
   TMR_StartBH_FansCO : TIMER := (PRE := 3000);   // Start Baghouse's Cleanout Timer
   TMR_StartHS : TIMER := (PRE := 3000);   // Run Hullers & Shellers Warning Timer
   TMR_StartPC1_Fans : TIMER := (PRE := 3000);   // Pre Clean Line 1 Fans Start Warning Timer
   TMR_StartPC1_FansCO : TIMER := (PRE := 3000);   // Pre Clean Line 1 Fans Cleanout Start Warning Timer
   TMR_StartPC2_Fans : TIMER := (PRE := 3000);   // Pre Clean Line 2 Fans Start Warning Timer
   TMR_StartPC2_FansCO : TIMER := (PRE := 3000);   // Pre Clean Line 2 Fans Cleanout Start Warning Timer
   TMR_StopBH1_Fans : TIMER := (PRE := 30000);   // Stop Baghouse 1 Fans Timer
   TMR_StopBH1_FansCo : TIMER := (PRE := 30000);   // Stop Baghouse 2 Fans Cleanout Timer
END_VAR

PROGRAM BagHouses   (* main routine BH_MainJSR *)
// BagHouses

ROUTINE BH_MainJSR   (* ladder *)
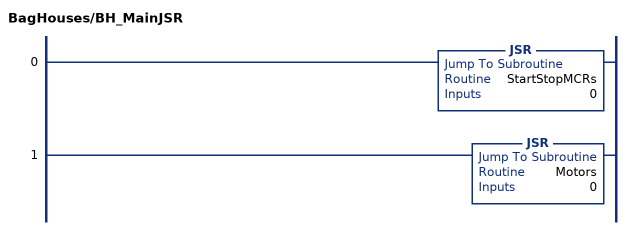
   0: JSR(StartStopMCRs,0);
   1: JSR(Motors,0);
END_ROUTINE

ROUTINE Motors   (* ladder *)
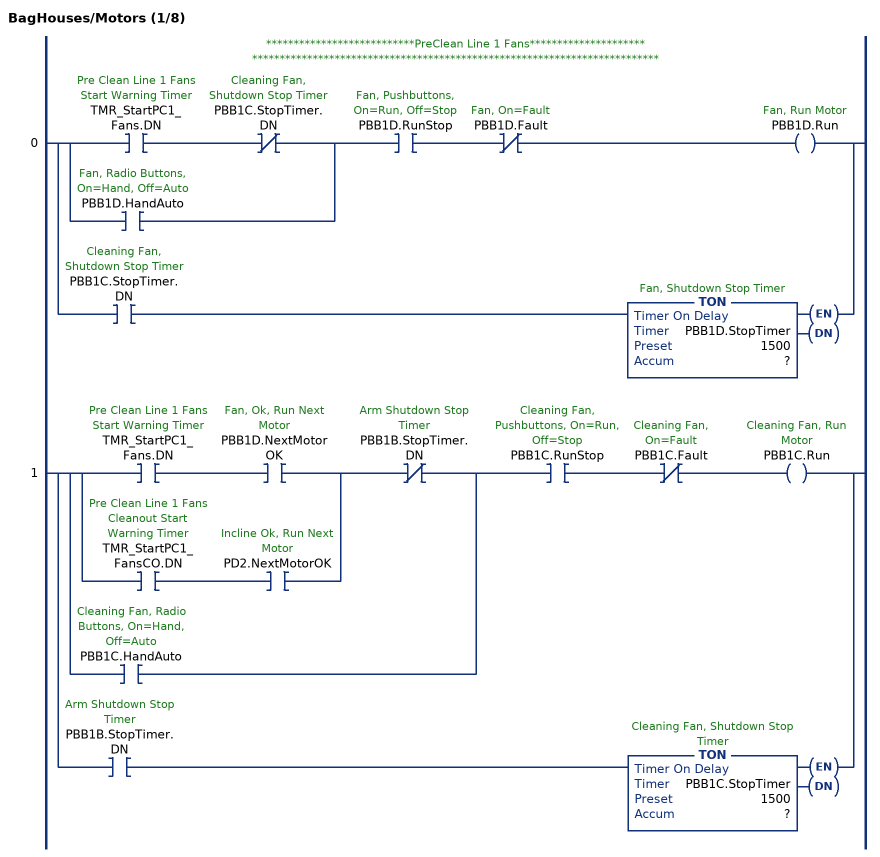
   // ***************************PreClean Line 1 Fans*********************
   // **************************************************************************
   0: [[XIC(TMR_StartPC1_Fans.DN) XIO(PBB1C.StopTimer.DN) ,XIC(PBB1D.HandAuto) ] XIC(PBB1D.RunStop) XIO(PBB1D.Fault) OTE(PBB1D.Run) ,XIC(PBB1C.StopTimer.DN) TON(PBB1D.StopTimer,?,?) ];
   1: [[[XIC(TMR_StartPC1_Fans.DN) XIC(PBB1D.NextMotorOK) ,XIC(TMR_StartPC1_FansCO.DN) XIC(PD2.NextMotorOK) ] XIO(PBB1B.StopTimer.DN) ,XIC(PBB1C.HandAuto) ] XIC(PBB1C.RunStop) XIO(PBB1C.Fault) OTE(PBB1C.Run) ,XIC(PBB1B.StopTimer.DN) TON(PBB1C.StopTimer,?,?) ];
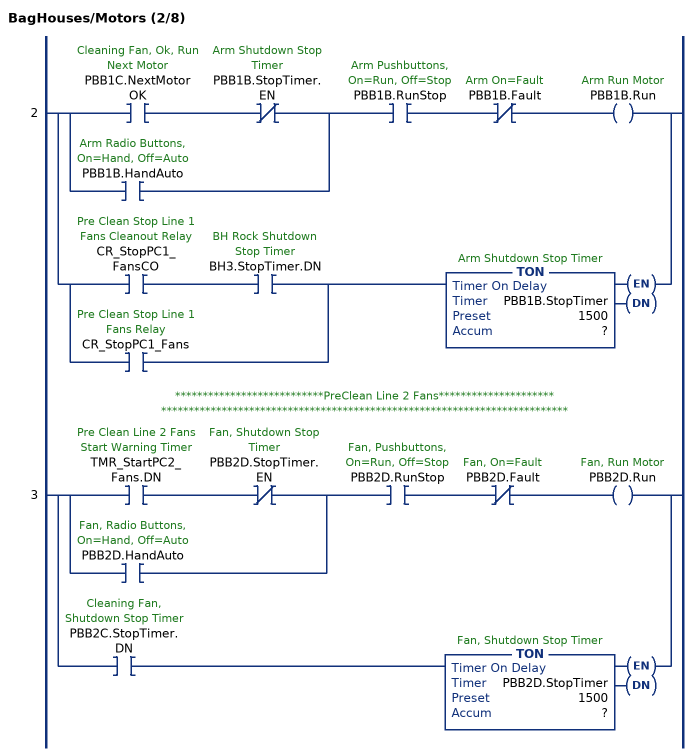
   2: [[XIC(PBB1C.NextMotorOK) XIO(PBB1B.StopTimer.EN) ,XIC(PBB1B.HandAuto) ] XIC(PBB1B.RunStop) XIO(PBB1B.Fault) OTE(PBB1B.Run) ,[XIC(CR_StopPC1_FansCO) XIC(BH3.StopTimer.DN) ,XIC(CR_StopPC1_Fans) ] TON(PBB1B.StopTimer,?,?) ];
   // ***************************PreClean Line 2 Fans*********************
   // **************************************************************************
   3: [[XIC(TMR_StartPC2_Fans.DN) XIO(PBB2D.StopTimer.EN) ,XIC(PBB2D.HandAuto) ] XIC(PBB2D.RunStop) XIO(PBB2D.Fault) OTE(PBB2D.Run) ,XIC(PBB2C.StopTimer.DN) TON(PBB2D.StopTimer,?,?) ];
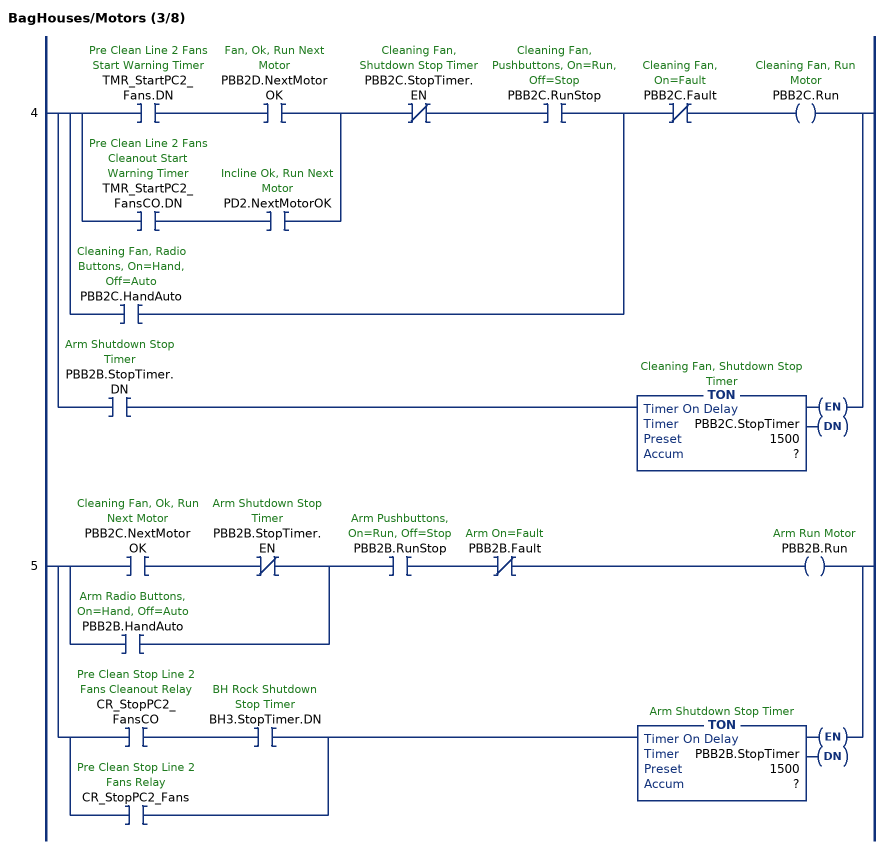
   4: [[[XIC(TMR_StartPC2_Fans.DN) XIC(PBB2D.NextMotorOK) ,XIC(TMR_StartPC2_FansCO.DN) XIC(PD2.NextMotorOK) ] XIO(PBB2C.StopTimer.EN) XIC(PBB2C.RunStop) ,XIC(PBB2C.HandAuto) ] XIO(PBB2C.Fault) OTE(PBB2C.Run) ,XIC(PBB2B.StopTimer.DN) TON(PBB2C.StopTimer,?,?) ];
   5: [[XIC(PBB2C.NextMotorOK) XIO(PBB2B.StopTimer.EN) ,XIC(PBB2B.HandAuto) ] XIC(PBB2B.RunStop) XIO(PBB2B.Fault) OTE(PBB2B.Run) ,[XIC(CR_StopPC2_FansCO) XIC(BH3.StopTimer.DN) ,XIC(CR_StopPC2_Fans) ] TON(PBB2B.StopTimer,?,?) ];
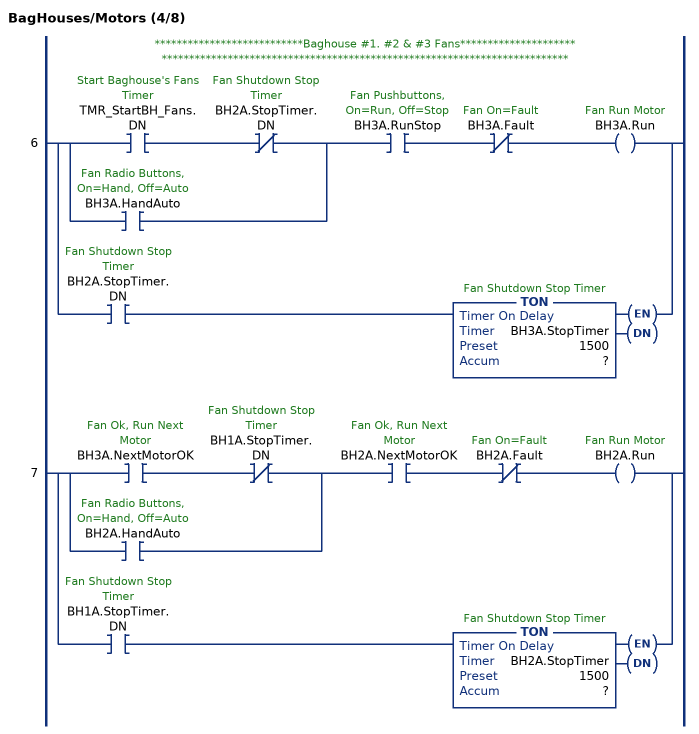
   // ***************************Baghouse #1. #2 & #3 Fans*********************
   // **************************************************************************
   6: [[XIC(TMR_StartBH_Fans.DN) XIO(BH2A.StopTimer.DN) ,XIC(BH3A.HandAuto) ] XIC(BH3A.RunStop) XIO(BH3A.Fault) OTE(BH3A.Run) ,XIC(BH2A.StopTimer.DN) TON(BH3A.StopTimer,?,?) ];
   7: [[XIC(BH3A.NextMotorOK) XIO(BH1A.StopTimer.DN) ,XIC(BH2A.HandAuto) ] XIC(BH2A.NextMotorOK) XIO(BH2A.Fault) OTE(BH2A.Run) ,XIC(BH1A.StopTimer.DN) TON(BH2A.StopTimer,?,?) ];
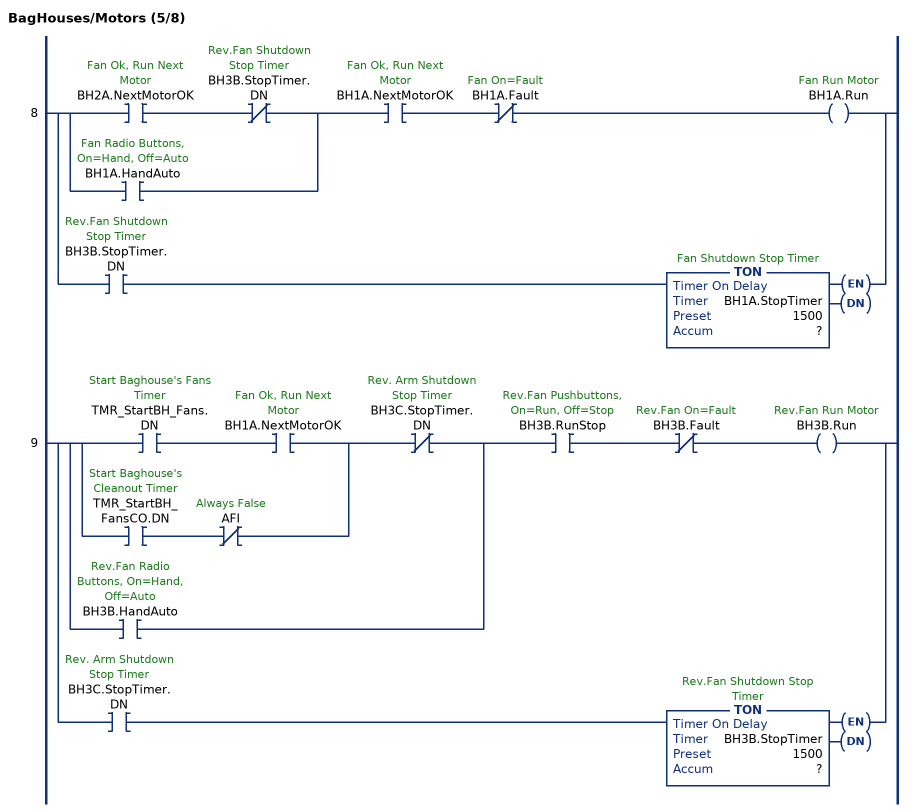
   8: [[XIC(BH2A.NextMotorOK) XIO(BH3B.StopTimer.DN) ,XIC(BH1A.HandAuto) ] XIC(BH1A.NextMotorOK) XIO(BH1A.Fault) OTE(BH1A.Run) ,XIC(BH3B.StopTimer.DN) TON(BH1A.StopTimer,?,?) ];
   9: [[[XIC(TMR_StartBH_Fans.DN) XIC(BH1A.NextMotorOK) ,XIC(TMR_StartBH_FansCO.DN) XIO(AFI) ] XIO(BH3C.StopTimer.DN) ,XIC(BH3B.HandAuto) ] XIC(BH3B.RunStop) XIO(BH3B.Fault) OTE(BH3B.Run) ,XIC(BH3C.StopTimer.DN) TON(BH3B.StopTimer,?,?) ];
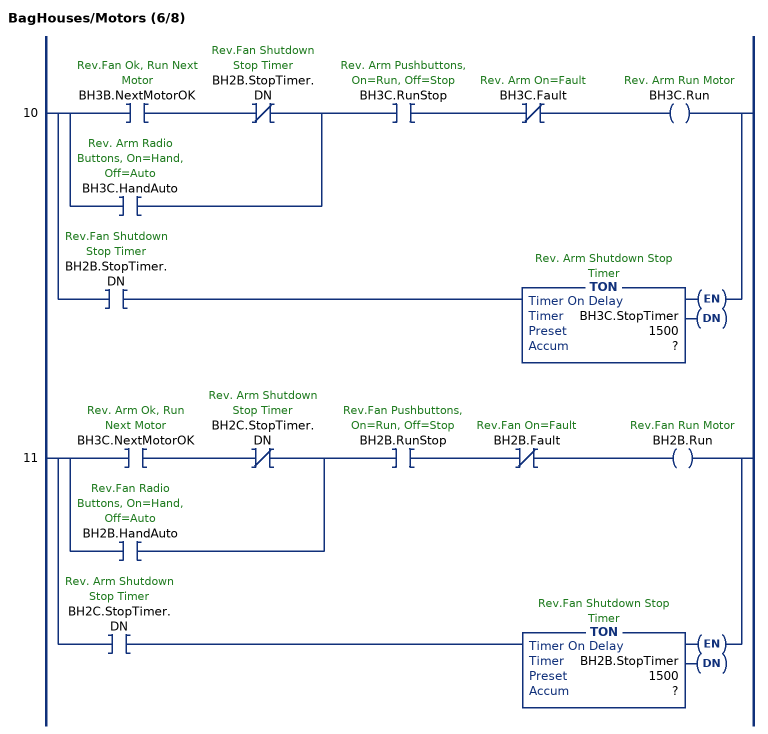
   10: [[XIC(BH3B.NextMotorOK) XIO(BH2B.StopTimer.DN) ,XIC(BH3C.HandAuto) ] XIC(BH3C.RunStop) XIO(BH3C.Fault) OTE(BH3C.Run) ,XIC(BH2B.StopTimer.DN) TON(BH3C.StopTimer,?,?) ];
   11: [[XIC(BH3C.NextMotorOK) XIO(BH2C.StopTimer.DN) ,XIC(BH2B.HandAuto) ] XIC(BH2B.RunStop) XIO(BH2B.Fault) OTE(BH2B.Run) ,XIC(BH2C.StopTimer.DN) TON(BH2B.StopTimer,?,?) ];
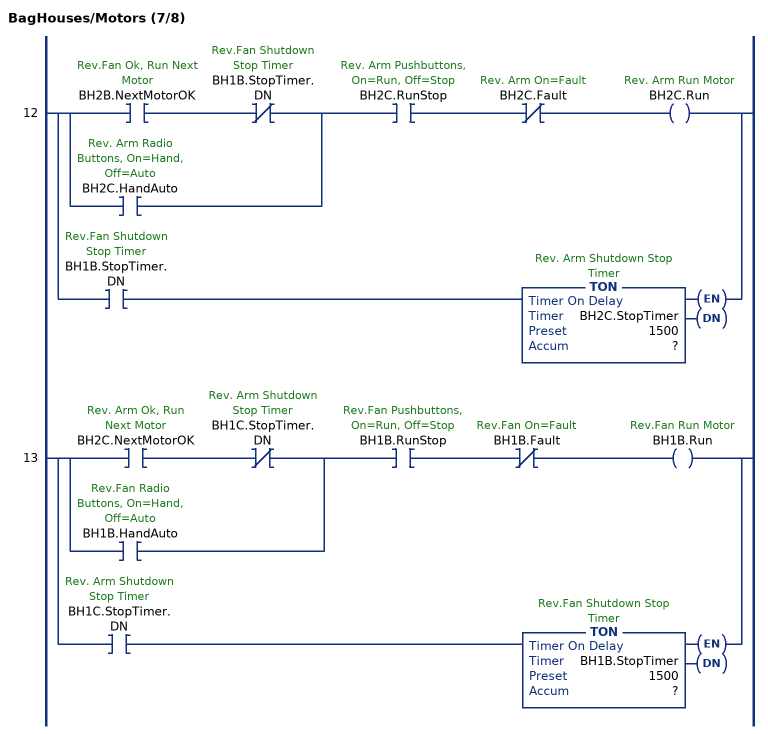
   12: [[XIC(BH2B.NextMotorOK) XIO(BH1B.StopTimer.DN) ,XIC(BH2C.HandAuto) ] XIC(BH2C.RunStop) XIO(BH2C.Fault) OTE(BH2C.Run) ,XIC(BH1B.StopTimer.DN) TON(BH2C.StopTimer,?,?) ];
   13: [[XIC(BH2C.NextMotorOK) XIO(BH1C.StopTimer.DN) ,XIC(BH1B.HandAuto) ] XIC(BH1B.RunStop) XIO(BH1B.Fault) OTE(BH1B.Run) ,XIC(BH1C.StopTimer.DN) TON(BH1B.StopTimer,?,?) ];
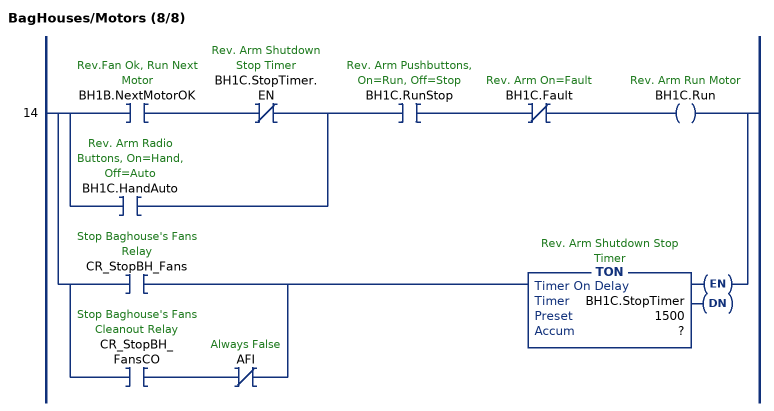
   14: [[XIC(BH1B.NextMotorOK) XIO(BH1C.StopTimer.EN) ,XIC(BH1C.HandAuto) ] XIC(BH1C.RunStop) XIO(BH1C.Fault) OTE(BH1C.Run) ,[XIC(CR_StopBH_Fans) ,XIC(CR_StopBH_FansCO) XIO(AFI) ] TON(BH1C.StopTimer,?,?) ];
END_ROUTINE

ROUTINE StartStopMCRs   (* ladder *)
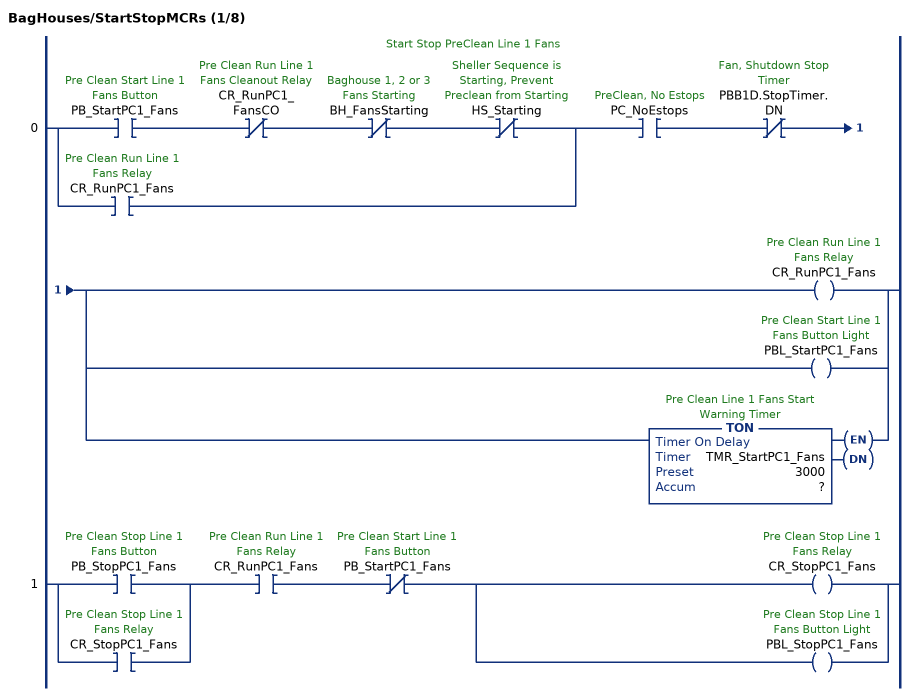
   // Start Stop PreClean Line 1 Fans
   0: [XIC(PB_StartPC1_Fans) XIO(CR_RunPC1_FansCO) XIO(BH_FansStarting) XIO(HS_Starting) ,XIC(CR_RunPC1_Fans) ]XIC(PC_NoEstops)XIO(PBB1D.StopTimer.DN)[OTE(CR_RunPC1_Fans) ,OTE(PBL_StartPC1_Fans) ,TON(TMR_StartPC1_Fans,?,?) ];
   1: [XIC(PB_StopPC1_Fans) ,XIC(CR_StopPC1_Fans) ]XIC(CR_RunPC1_Fans)XIO(PB_StartPC1_Fans)[OTE(CR_StopPC1_Fans) ,OTE(PBL_StopPC1_Fans) ];
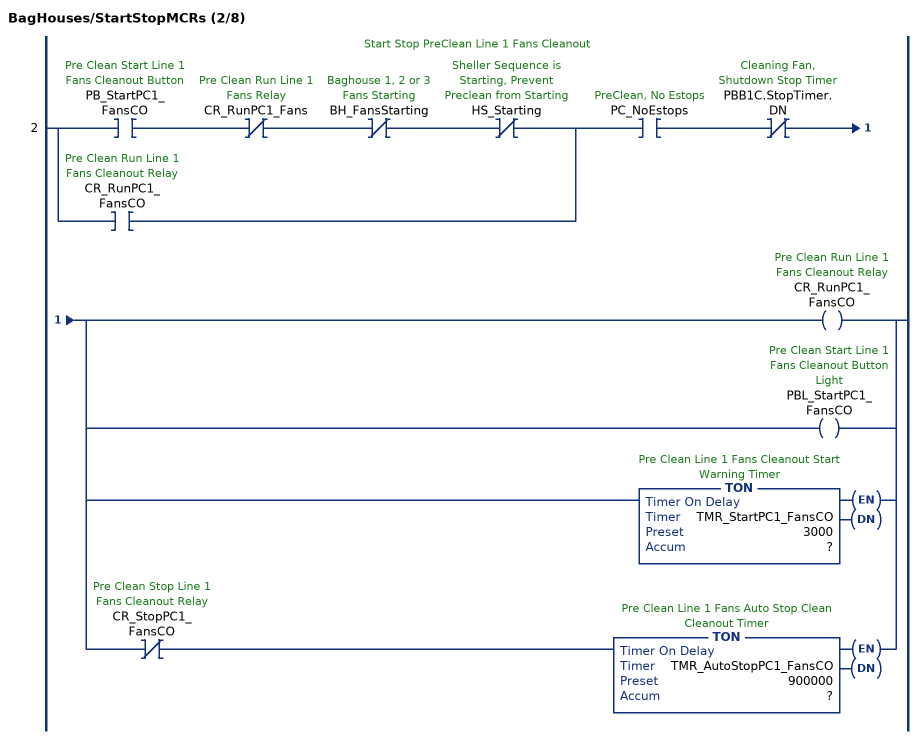
   // Start Stop PreClean Line 1 Fans Cleanout
   2: [XIC(PB_StartPC1_FansCO) XIO(CR_RunPC1_Fans) XIO(BH_FansStarting) XIO(HS_Starting) ,XIC(CR_RunPC1_FansCO) ]XIC(PC_NoEstops)XIO(PBB1C.StopTimer.DN)[OTE(CR_RunPC1_FansCO) ,OTE(PBL_StartPC1_FansCO) ,TON(TMR_StartPC1_FansCO,?,?) ,XIO(CR_StopPC1_FansCO) TON(TMR_AutoStopPC1_FansCO,?,?) ];
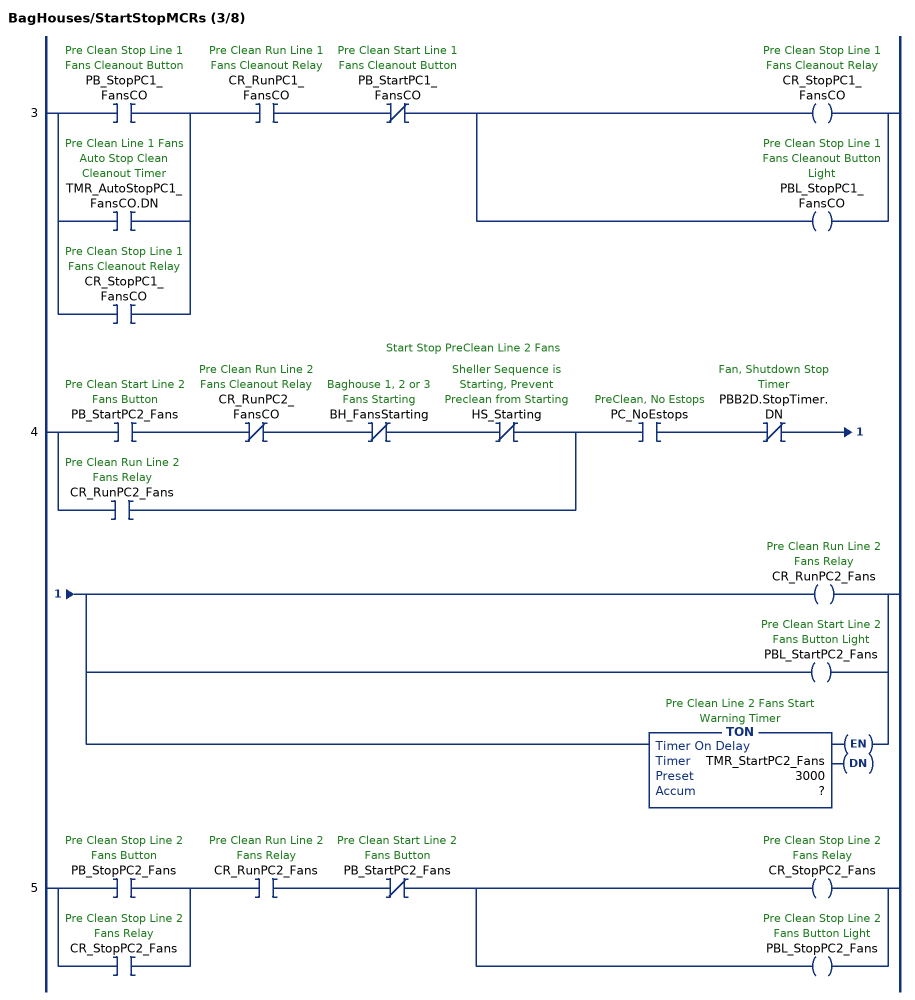
   3: [XIC(PB_StopPC1_FansCO) ,XIC(TMR_AutoStopPC1_FansCO.DN) ,XIC(CR_StopPC1_FansCO) ]XIC(CR_RunPC1_FansCO)XIO(PB_StartPC1_FansCO)[OTE(CR_StopPC1_FansCO) ,OTE(PBL_StopPC1_FansCO) ];
   // Start Stop PreClean Line 2 Fans
   4: [XIC(PB_StartPC2_Fans) XIO(CR_RunPC2_FansCO) XIO(BH_FansStarting) XIO(HS_Starting) ,XIC(CR_RunPC2_Fans) ]XIC(PC_NoEstops)XIO(PBB2D.StopTimer.DN)[OTE(CR_RunPC2_Fans) ,OTE(PBL_StartPC2_Fans) ,TON(TMR_StartPC2_Fans,?,?) ];
   5: [XIC(PB_StopPC2_Fans) ,XIC(CR_StopPC2_Fans) ]XIC(CR_RunPC2_Fans)XIO(PB_StartPC2_Fans)[OTE(CR_StopPC2_Fans) ,OTE(PBL_StopPC2_Fans) ];
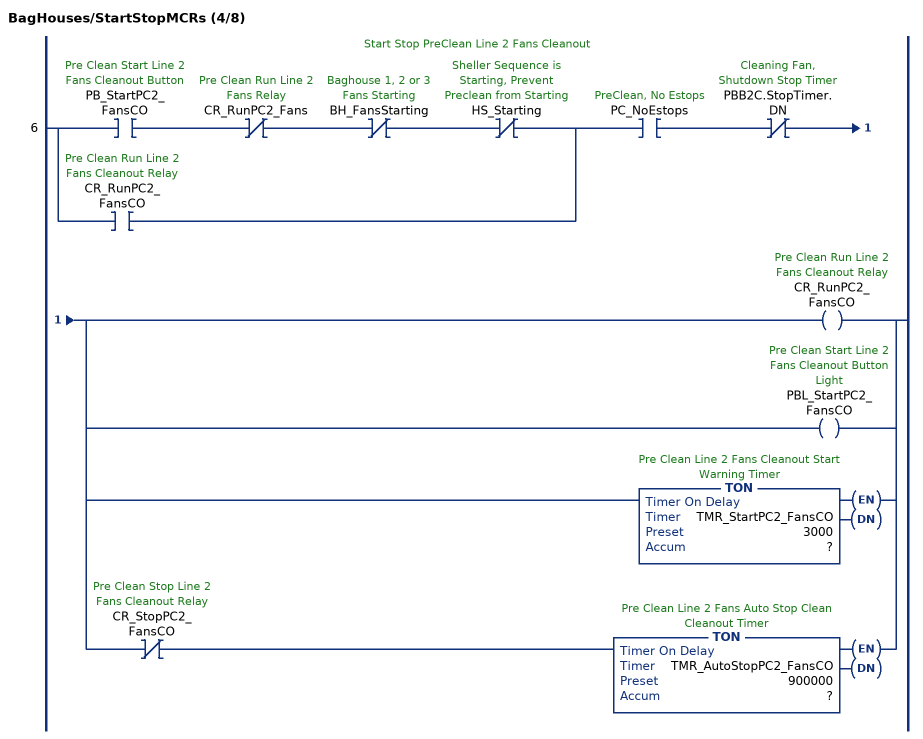
   // Start Stop PreClean Line 2 Fans Cleanout
   6: [XIC(PB_StartPC2_FansCO) XIO(CR_RunPC2_Fans) XIO(BH_FansStarting) XIO(HS_Starting) ,XIC(CR_RunPC2_FansCO) ]XIC(PC_NoEstops)XIO(PBB2C.StopTimer.DN)[OTE(CR_RunPC2_FansCO) ,OTE(PBL_StartPC2_FansCO) ,TON(TMR_StartPC2_FansCO,?,?) ,XIO(CR_StopPC2_FansCO) TON(TMR_AutoStopPC2_FansCO,?,?) ];
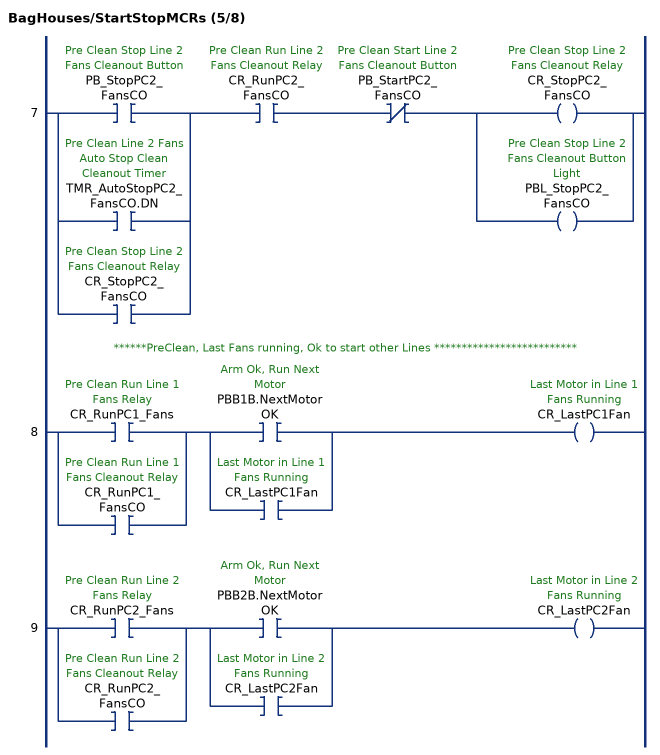
   7: [XIC(PB_StopPC2_FansCO) ,XIC(TMR_AutoStopPC2_FansCO.DN) ,XIC(CR_StopPC2_FansCO) ]XIC(CR_RunPC2_FansCO)XIO(PB_StartPC2_FansCO)[OTE(CR_StopPC2_FansCO) ,OTE(PBL_StopPC2_FansCO) ];
   // ******PreClean, Last Fans running, Ok to start other Lines **************************
   8: [XIC(CR_RunPC1_Fans) ,XIC(CR_RunPC1_FansCO) ][XIC(PBB1B.NextMotorOK) ,XIC(CR_LastPC1Fan) ]OTE(CR_LastPC1Fan);
   9: [XIC(CR_RunPC2_Fans) ,XIC(CR_RunPC2_FansCO) ][XIC(PBB2B.NextMotorOK) ,XIC(CR_LastPC2Fan) ]OTE(CR_LastPC2Fan);
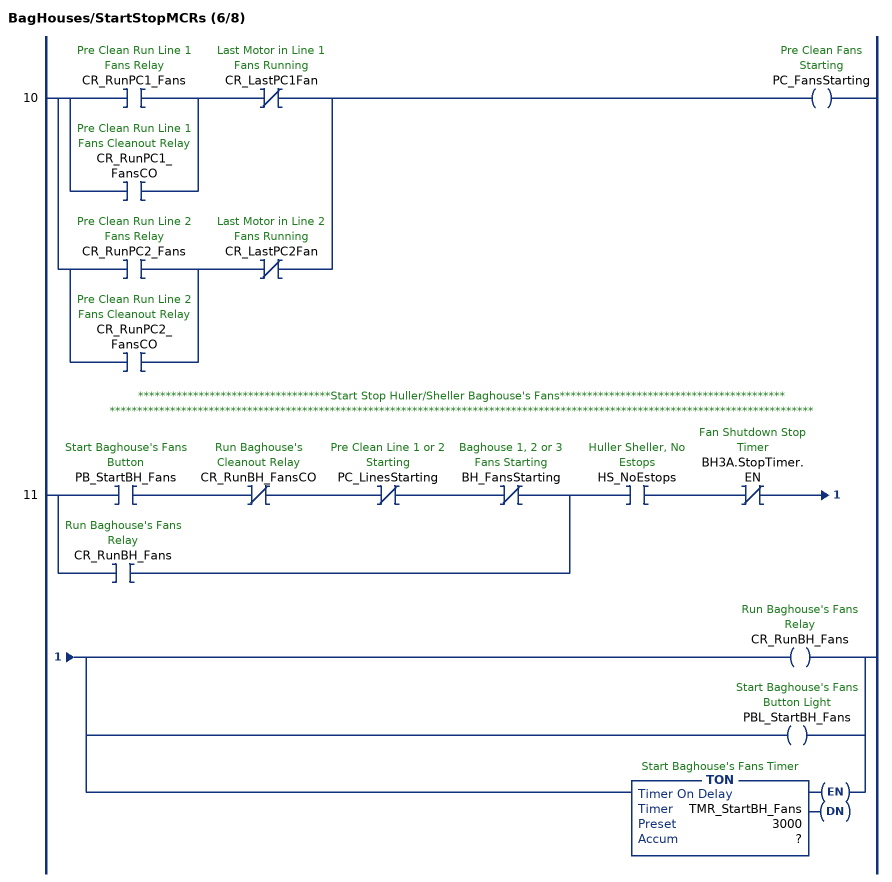
   10: [[XIC(CR_RunPC1_Fans) ,XIC(CR_RunPC1_FansCO) ] XIO(CR_LastPC1Fan) ,[XIC(CR_RunPC2_Fans) ,XIC(CR_RunPC2_FansCO) ] XIO(CR_LastPC2Fan) ]OTE(PC_FansStarting);
   // ***********************************Start Stop Huller/Sheller Baghouse's Fans*****************************************
   // ********************************************************************************************************************************
   11: [XIC(PB_StartBH_Fans) XIO(CR_RunBH_FansCO) XIO(PC_LinesStarting) XIO(BH_FansStarting) ,XIC(CR_RunBH_Fans) ]XIC(HS_NoEstops)XIO(BH3A.StopTimer.EN)[OTE(CR_RunBH_Fans) ,OTE(PBL_StartBH_Fans) ,TON(TMR_StartBH_Fans,?,?) ];
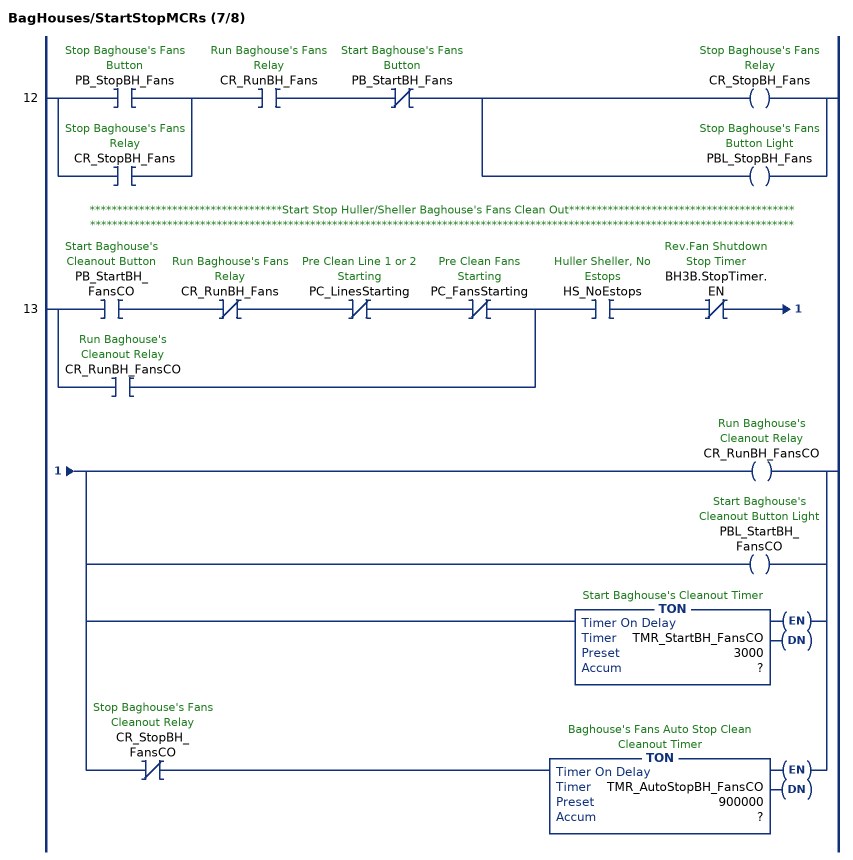
   12: [XIC(PB_StopBH_Fans) ,XIC(CR_StopBH_Fans) ]XIC(CR_RunBH_Fans)XIO(PB_StartBH_Fans)[OTE(CR_StopBH_Fans) ,OTE(PBL_StopBH_Fans) ];
   // ***********************************Start Stop Huller/Sheller Baghouse's Fans Clean Out*****************************************
   // ********************************************************************************************************************************
   13: [XIC(PB_StartBH_FansCO) XIO(CR_RunBH_Fans) XIO(PC_LinesStarting) XIO(PC_FansStarting) ,XIC(CR_RunBH_FansCO) ]XIC(HS_NoEstops)XIO(BH3B.StopTimer.EN)[OTE(CR_RunBH_FansCO) ,OTE(PBL_StartBH_FansCO) ,TON(TMR_StartBH_FansCO,?,?) ,XIO(CR_StopBH_FansCO) TON(TMR_AutoStopBH_FansCO,?,?) ];
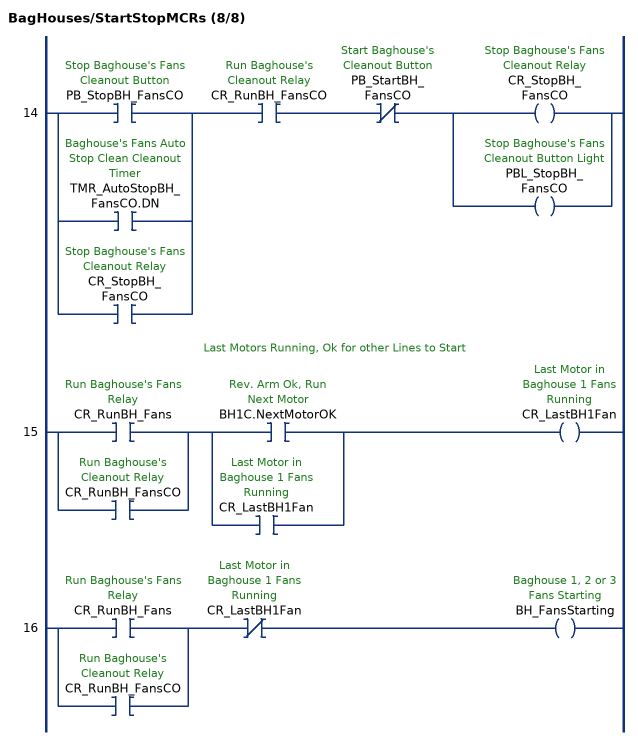
   14: [XIC(PB_StopBH_FansCO) ,XIC(TMR_AutoStopBH_FansCO.DN) ,XIC(CR_StopBH_FansCO) ]XIC(CR_RunBH_FansCO)XIO(PB_StartBH_FansCO)[OTE(CR_StopBH_FansCO) ,OTE(PBL_StopBH_FansCO) ];
   // Last Motors Running, Ok for other Lines to Start
   15: [XIC(CR_RunBH_Fans) ,XIC(CR_RunBH_FansCO) ][XIC(BH1C.NextMotorOK) ,XIC(CR_LastBH1Fan) ]OTE(CR_LastBH1Fan);
   16: [XIC(CR_RunBH_Fans) ,XIC(CR_RunBH_FansCO) ]XIO(CR_LastBH1Fan)OTE(BH_FansStarting);
END_ROUTINE
END_PROGRAM

PROGRAM HullerSheller   (* main routine HS_MainJSR *)
VAR
   CTR_HornBeeps : COUNTER := (PRE := 3);   // Number of times horn beeps
   FaultPresent : BOOL;   // A Huller-Sheller Fault is Present
   FaultReset : BOOL;   // Huller-Sheller Fault Reset
   HS_AlarmPulseHorn : BOOL;   // Huller Sheller, New Alarm, Pulse Horn
   HS_FaultResetHorn : BOOL;   // Hullwe Sheller, Fault Reset, sound Horn
   NewFault : BOOL;   // New Huller-Sheller Fault has just occured
   NewFaultBeepHorn : BOOL;   // NewFault or Warning, Pulse Horn
   NewWarning : BOOL;   // New Huller-Sheller Warning has just occured
   Num_Faults : DINT;   // Number of Huller-Sheller Faults
   Num_Faults_LS : DINT;   // Number of Huller-Sheller Faults Last PLC Scan
   Num_Warning_LS : DINT;   // Number of Huller-Sheller Warnings Last Scan, Detect New
   Num_Warnings : DINT;   // Number of Huller-Sheller Warnings
   Reset_TOF_PRE : DINT;   // Reset pulse duration to Drives
   SpeedIsFactored : BOOL;   // Speed of VFD is factored by Master Speed Factor
   TempAlarm : BOOL;   // Temp Motor has Alarm
   TempAtSpeed : BOOL;   // Temp Motor is At Speed
   TempCommAlarm : BOOL;   // Temp Motor, AOP communications Alarm
   TempDecelerating : BOOL;   // Temp Motor is Decelerating
   TempFaulted : BOOL;   // Temp Motor is Faulted
   TempImbalanceTrip : BOOL;   // Temp Motor, Phase Imbalance Trip
   TempImbalanceWarning : BOOL;   // Temp Motor, Phase Imbalance Warning
   TempMotor : Motor := (Fault_TON.PRE := 1000, Warning_TON.PRE := 1000, Reset_TOF.PRE := 500); {access None}   // Temp Motor Tag for Subroutines
   TempMotor1 : Motor := (Fault_TON.PRE := 1000, Warning_TON.PRE := 1000, Reset_TOF.PRE := 500); {access None}
   TempOL_Percent : DINT;   // Temp Motor Percent Overload
   TempOverloadTrip : BOOL;   // Temp Motor, Overload Trip
   TempOverloadWarning : BOOL;   // Temp Motor, Overlaod Warning
   TempPhaseLossTrip : BOOL;   // Temp Motor, Phase Loss Trip
   TempReady : BOOL;   // Temp Motor is ready
   TempRunning : BOOL;   // Temp Motor is Running
   TempTriped : BOOL;   // Temp Motor Tripped
   TempVFD : VFD_Extra;   // Temp VFD Structure
   TempWarning : BOOL;   // Temp Motor Warning
   TMR_HornFlasher : TIMER := (PRE := 1000);   // Fault Horn Flasher timer
   TMR_HS_FaultResetHorn : TIMER := (PRE := 3000);   // Huller Sheller, Fault Reset, sound Horn
END_VAR

ROUTINE Alarms   (* ladder *)
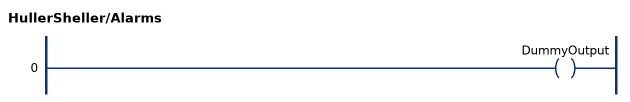
   0: OTE(DummyOutput);
END_ROUTINE
